INTERFACE Imotor

PROPERTY error : bool
GET
END_GET
SET
END_SET
END_PROPERTY

METHOD run : BOOL
END_METHOD

PROPERTY running : bool
GET
END_GET
SET
END_SET
END_PROPERTY

METHOD status : BOOL
END_METHOD

METHOD stop : BOOL
VAR_INPUT
END_VAR
END_METHOD

END_INTERFACE

(* stored: Version 1.1.0.1, ProductVersion 3.1.4024.12
   Itf Imotor: Id {75a4f806-4e53-43be-b637-b05eaf11f7ef}
   Property error: Id {7574cc5d-08be-4d25-9e18-c7f725a5c3ee}
   Get Get: Id {66504c63-cf26-4f66-8dab-32209f94ce5c}
   Set Set: Id {6fbc2fc2-bcfa-4ac8-913c-48b1b3df2894}
   Method run: Id {aba3c462-42c5-4efe-981f-4971d8d236c5}
   Property running: Id {4f14fadd-fc2e-433d-84eb-c6ff3a2dcbfe}
   Get Get: Id {9ad8f65e-97a6-4abe-897c-c98837dead15}
   Set Set: Id {04fc6342-18e5-414c-8809-9ea184f16158}
   Method status: Id {2dcb4e3a-65cc-499d-ab4f-66ebed2dfccd}
   Method stop: Id {a00217d8-133a-4b2c-85e8-55e9900fe693} *)
